{attribute 'qualified_only'}
{attribute 'strict'}
{attribute 'to_string'}
TYPE Betriebszustand :
(
	Aus,
	Produktion,
	Fehler,
	Warnung,
	Init,
	Bereit,
	Fertig
);
END_TYPE

(* stored: Version 1.1.0.1
   DUT Betriebszustand: Id {dae00368-c1d9-4def-aba5-b7ba5fdd79cf} *)
